{attribute 'TcGenerated'}
{attribute 'no-analysis'}
{attribute 'linkalways'}
// This function has been automatically generated from the project information.
VAR_GLOBAL CONSTANT
	{attribute 'const_non_replaced'}
	stLibVersion_Tc3_LmDualAxisCoordinator : ST_LibVersion := (iMajor := 1, iMinor := 0, iBuild := 0, iRevision := 0, nFlags := 0, sVersion := '1.0.0.0');
END_VAR

(* stored: Version 1.1.0.1, ProductVersion 3.1.4026.18
   GVL Global_Version: Id {fd81003c-48fd-4aeb-93c8-474496817c5c} *)
